FUNCTION_BLOCK FB_Example
VAR
    x : INT;
END_VAR
BEGIN // start of code
y := 1;
END_FUNCTION_BLOCK
